(* IEC 61131-3 sources: IEC61131-3-CDSV3/Math Expressions Evaluator/src/20 Program Organization Units/Low Level, 3 files *)

(* ---- FuEvaluateExpression.pou ---- *)
(*#-#-#-#-#-#-#-#-#-#---Declaration---#-#-#-#-#-#-#-#-#-#-#-#-#*)

// Evaluates the expression.
// All expressions use LREAL as data type for operations, which is also the result output.
//
// The following math operation behaviour applies:
//  - In general: If any of the operands is a special value (+Inf, -Inf, NaN), then an error is returned
//  - For Division (/): Division by zero yields depending on ParameterList.eDivisionByZero into an error or not
//  - For Modulo (%): Both operands are converted to LINT and the result is converted back to LREAL
//
// The return value will indicate a successful evaluation.
{attribute 'qualified_only'}
FUNCTION FuEvaluateExpression : BOOL
VAR_INPUT
    typExpressionSteps: typExpressionOperationSteps;   // The expression providing steps for complex terms
    alrVariables: ARRAY [*] OF LREAL;                  // Variables to use
END_VAR
VAR_OUTPUT
    lrResult: LREAL;                                   // Result output
    sError: STRING;                                    // Error message
END_VAR
{library PRIVATE}
VAR
    i: UINT;
    tempResult: LREAL;
    tempError: STRING;

    tempInternalVariables: ARRAY [0..ParameterList.uiMaxInternalVars] OF LREAL;
END_VAR
(*#-#-#-#-#-#-#-#-#-#---Implementation---#-#-#-#-#-#-#-#-#-#-#-#-#*)

IF typExpressionSteps.uiCountSteps = 0 THEN
    FuEvaluateExpression := TRUE;
    RETURN;
END_IF

FOR i := 0 TO (typExpressionSteps.uiCountSteps - 1) BY 1 DO
    IF NOT FuEvaluateStep(typExpressionSteps.atSteps[i],  alrVariables, tempInternalVariables, lrResult => tempResult, sError => tempError) THEN
        sError := tempError;
        RETURN;
    END_IF

    // Always have the result in internal variable 0
    tempInternalVariables[0] := tempResult;

    IF
        typExpressionSteps.atSteps[i].uiInternalVariableTarget > 0 AND_THEN
        typExpressionSteps.atSteps[i].uiInternalVariableTarget >= 1 AND_THEN
        typExpressionSteps.atSteps[i].uiInternalVariableTarget <= ParameterList.uiMaxInternalVars
    THEN
        tempInternalVariables[typExpressionSteps.atSteps[i].uiInternalVariableTarget] := tempResult;
    END_IF
END_FOR

lrResult := tempResult;
FuEvaluateExpression := TRUE;

(* ---- FuStepizeExpression.pou ---- *)
(*#-#-#-#-#-#-#-#-#-#---Declaration---#-#-#-#-#-#-#-#-#-#-#-#-#*)

// Turns a tokenized expression into a stepized expression,
// providing steps for each "group" operation to be done,
// including taking care of ordering.
//
// Group operations include function calls and expressions inside ().
// Operations such as "1 + 5 - 2" are not split up and
// are evaluated left to right from the evaluator.
//
// The return value signifies whether the operation has been successfully completed.
// This function should only return false, when we run out of internal variables
// or there are no tokens.
{attribute 'qualified_only'}
FUNCTION FuStepizeExpression : BOOL
VAR_INPUT
    typTokenExpression: typTokenizedExpression;
END_VAR
VAR_OUTPUT
    typSteps: typExpressionOperationSteps;
END_VAR
{library PRIVATE}
VAR
    i: UINT;
    j: UINT;

    tempEndTokenIndex: UINT;
END_VAR
VAR // Data used throughout each loop iteration
    tempFoundGroups: ARRAY [0..ParameterList.uiMaxExpressionTokens] OF typStepizeGroupFound;
    tempCountFoundGroups: UINT;

    tempFoundGroupsTokens: ARRAY [0..ParameterList.uiMaxExpressionTokens] OF typExpressionToken;
    tempCountFoundGroupsTokens: UINT;

    tempLastStartedGroups: ARRAY [0..ParameterList.uiMaxExpressionTokens] OF UINT;
    tempCountLastStartedGroups: UINT;
END_VAR
VAR CONSTANT
    {warning disable C0228}
    INVALID_TOKEN: typExpressionToken := (eType := eTokenType.INVALID);
    EMPTY_TOKEN_ARR: ARRAY [0..ParameterList.uiMaxExpressionTokens] OF typExpressionToken;
    {warning restore C0228}
END_VAR
(*#-#-#-#-#-#-#-#-#-#---Implementation---#-#-#-#-#-#-#-#-#-#-#-#-#*)

IF typTokenExpression.uiCountTokens = 0 THEN
    RETURN;
END_IF

// Step 1: Find each group and make a list out of it
FOR i := 0 TO (typTokenExpression.uiCountTokens - 1) BY 1 DO
    IF
        typTokenExpression.atTokens[i].eType = eTokenType.GROUP_START OR_ELSE
        typTokenExpression.atTokens[i].eType = eTokenType.FUNCTION_CALL
    THEN
        tempFoundGroups[tempCountFoundGroups].uiTokenIndex := i;
        tempFoundGroups[tempCountFoundGroups].uiGroupNumber := typTokenExpression.atTokens[i].uiGroupNumber;

        tempCountFoundGroups := tempCountFoundGroups + 1;
    END_IF
END_FOR

// Skip step 2 and 3 if we found NO groups
IF tempCountFoundGroups > 0 THEN
    // Step 2: Sort the found groups array by group number and then token index
    FuInsertSortStepizeGroupFound(ADR(tempFoundGroups), tempCountFoundGroups);

    // Step 3: Consume found groups, take the tokens and insert ASSIGN_INTERNAL_VAR tokens
    //         -> Note: The found groups index + 1 corresponds to the internal variable number
    FOR i := 0 TO (tempCountFoundGroups - 1) BY 1 DO
        tempFoundGroupsTokens := EMPTY_TOKEN_ARR;
        tempCountFoundGroupsTokens := 0;

        tempCountLastStartedGroups := 0;
        tempEndTokenIndex := 0;

        FOR j := tempFoundGroups[i].uiTokenIndex TO (typTokenExpression.uiCountTokens - 1) BY 1 DO
            IF typTokenExpression.atTokens[j].eType = eTokenType.INVALID THEN
                CONTINUE;
            END_IF

            IF typTokenExpression.atTokens[j].eType = eTokenType.GROUP_START AND_THEN typTokenExpression.atTokens[j].uiGroupNumber <> tempFoundGroups[i].uiGroupNumber THEN
                // Another group started, we need to ignore those tokens now
                tempLastStartedGroups[tempCountLastStartedGroups] := typTokenExpression.atTokens[j].uiGroupNumber;
                tempCountLastStartedGroups := tempCountLastStartedGroups + 1;

                CONTINUE;
            ELSIF
                typTokenExpression.atTokens[j].eType = eTokenType.GROUP_END AND_THEN
                tempCountLastStartedGroups > 0 AND_THEN
                typTokenExpression.atTokens[j].uiGroupNumber = tempLastStartedGroups[(tempCountLastStartedGroups - 1)]
            THEN
                // Another group ended, we can now start caring again, if the count drops to 0
                tempCountLastStartedGroups := tempCountLastStartedGroups - 1;

                CONTINUE; // Taking care of using the internal variable of each group will be done later using "tempSkipTokenHints"
            ELSIF tempCountLastStartedGroups > 0 THEN
                // As long as another group are still open, prevent the other two clauses (the elsif and else) from being able to execute
                CONTINUE;
            END_IF

            IF typTokenExpression.atTokens[j].eType = eTokenType.GROUP_END AND_THEN typTokenExpression.atTokens[j].uiGroupNumber = tempFoundGroups[i].uiGroupNumber THEN
                // We've reached the end of our group, stop taking tokens away, add a hint for later about skipping tokens, and exit this loop
                tempEndTokenIndex := j;
                EXIT;
            ELSIF typTokenExpression.atTokens[j].eType = eTokenType.GROUP_START AND_THEN typTokenExpression.atTokens[j].uiGroupNumber = tempFoundGroups[i].uiGroupNumber THEN
                // Ignore group starts of ourself (we dont need those tokens)
                CONTINUE;
            END_IF

            IF typTokenExpression.atTokens[j].eType = eTokenType.FUNCTION_CALL_END AND_THEN typTokenExpression.atTokens[j].uiGroupNumber = tempFoundGroups[i].uiGroupNumber THEN
                // We've reached the end of our group, stop taking tokens away, add a hint for later about skipping tokens, and exit this loop
                tempEndTokenIndex := j;
                EXIT;
            END_IF

            tempFoundGroupsTokens[tempCountFoundGroupsTokens] := typTokenExpression.atTokens[j];
            tempCountFoundGroupsTokens := tempCountFoundGroupsTokens + 1;
        END_FOR

        typSteps.atSteps[typSteps.uiCountSteps].atTokens := tempFoundGroupsTokens;
        typSteps.atSteps[typSteps.uiCountSteps].uiCountTokens := tempCountFoundGroupsTokens;
        typSteps.atSteps[typSteps.uiCountSteps].uiInternalVariableTarget := i + 1;

        IF i >= ParameterList.uiMaxInternalVars THEN
            FuStepizeExpression := FALSE;
            RETURN;
        END_IF

        // Replace all tokens with invalid tokens, if necessary, the first token will be replaced with INTERNAL_VAR
        FOR j := tempFoundGroups[i].uiTokenIndex TO tempEndTokenIndex BY 1 DO
            typTokenExpression.atTokens[j] := INVALID_TOKEN;
        END_FOR

        IF tempFoundGroups[i].uiTokenIndex = 0 AND_THEN tempEndTokenIndex = (typTokenExpression.uiCountTokens - 1) THEN
            ;// Do not generate internal var token, because all tokens are covered
        ELSE
            // Rewrite tokens and replace them with one INTERNAL_VAR and INVALID tokens
            typTokenExpression.atTokens[tempFoundGroups[i].uiTokenIndex] := INVALID_TOKEN;
            typTokenExpression.atTokens[tempFoundGroups[i].uiTokenIndex].eType := eTokenType.INTERNAL_VAR;
            typTokenExpression.atTokens[tempFoundGroups[i].uiTokenIndex].lrValue := TO_LREAL((i + 1));
        END_IF

        typSteps.uiCountSteps := typSteps.uiCountSteps + 1;
    END_FOR
END_IF

// Step 4: Rewrite the tokens, skip INVALID tokens
FOR i := 0 TO (typTokenExpression.uiCountTokens - 1) BY 1 DO
    IF typTokenExpression.atTokens[i].eType = eTokenType.INVALID THEN
        CONTINUE;
    END_IF

    j := typSteps.atSteps[typSteps.uiCountSteps].uiCountTokens;

    typSteps.atSteps[typSteps.uiCountSteps].atTokens[j] := typTokenExpression.atTokens[i];
    typSteps.atSteps[typSteps.uiCountSteps].uiCountTokens := j + 1;
END_FOR

IF typSteps.atSteps[typSteps.uiCountSteps].uiCountTokens > 0 THEN
    typSteps.uiCountSteps := typSteps.uiCountSteps + 1;
END_IF

// Step 5: Profit, each step should now contain a particular operation set
// Note: Operations as "1 + 5 + 6" are handled inline in the evaluator, since the result of the previous op "1 + 5" can be used as "$result + 5"
FuStepizeExpression := TRUE;

(* ---- FuTokenizeExpression.pou ---- *)
(*#-#-#-#-#-#-#-#-#-#---Declaration---#-#-#-#-#-#-#-#-#-#-#-#-#*)

// Tokenizes a given math expression into a stream of tokens.
// The return value signifies whether tokenization was successful,
// or during tokenization an invalid expression was encountered.
// Please note, during tokenization not all error cases are checked.
{attribute 'qualified_only'}
FUNCTION FuTokenizeExpression : BOOL
VAR_INPUT
    sExpression: STRING(255);                 // The expression string to tokenize
END_VAR
VAR_OUTPUT
    typExpression: typTokenizedExpression;    // The tokenized expression
    sError: STRING;                           // Error message
END_VAR
{library PRIVATE}
VAR
    i: UINT;
    j: UINT;

    tempChar: BYTE;
    tempNextChar: BYTE;

    tempFunEndDetected: BOOL;
END_VAR
VAR // Data used throughout each loop iteration
    tempIndex: UINT;

    tempIdentifierStr: STRING(5);
    tempPtrByte: POINTER TO BYTE;

    tempVarOpen: BOOL;

    tempGroupOpen: INT := 0;
    tempGroupNum: UINT := 50;

    tempFunOpen: BOOL;
    tempFunIndex: UINT;
    tempFunArgsCount: UINT;

    tempNumOpen: BOOL;
    tempNumSign: BOOL; // TRUE = negative

    tempValueStr: STRING(80);
END_VAR
(*#-#-#-#-#-#-#-#-#-#---Implementation---#-#-#-#-#-#-#-#-#-#-#-#-#*)

IF sExpression = '' THEN
    sError := 'Empty expression';
    RETURN;
END_IF

sError := '';

// Assert a clean string (CODESYS does not assert that the whole string contains NUL bytes, only sets the first byte as NUL byte!)
// tempValueStr is VAR_TEMP and should get completely initialized as an empty string (all bytes = NUL), but the truth is the memory space
// gets reused and thus leftovers from the previous execution can be left there, since only the first byte is set to NUL
// (which is described by CODESYS as "new initialization", which is technically wrong!)
FOR i := 0 TO SIZEOF(tempValueStr) BY 1 DO
    tempValueStr[i] := 0;
END_FOR

FOR i := 0 TO 255 BY 1 DO
    IF sExpression[i] = 0 THEN
        EXIT;
    ELSIF tempIndex > ParameterList.uiMaxExpressionTokens THEN
        sError := 'Too many expressions';
        EXIT;
    END_IF

    tempIdentifierStr := '';
    tempPtrByte := 0;

    tempChar := sExpression[i];

    CASE tempChar OF
        Constants.CHAR_WHITESPACE, Constants.CHAR_NEWLINE, Constants.CHAR_CAR_RETURN:
            IF tempNumOpen THEN
                typExpression.atTokens[tempIndex].eType := eTokenType.NUMBER;
                typExpression.atTokens[tempIndex].lrValue := STRING_TO_LREAL(tempValueStr);

                tempValueStr := '';
                tempNumOpen := FALSE;
            ELSIF tempVarOpen THEN
                typExpression.atTokens[tempIndex].eType := eTokenType.VARIABLE;
                typExpression.atTokens[tempIndex].lrValue := STRING_TO_LREAL(tempValueStr);

                tempValueStr := '';
                tempVarOpen := FALSE;
            ELSE
                CONTINUE; // Ignore whitespace, newline (\n) and carriage return (\r)
            END_IF

        Constants.CHAR_VARIABLE:
            IF tempVarOpen OR_ELSE tempNumOpen THEN
                sError := Standard.CONCAT('Unexpected VARIABLE "\" start at token ', TO_STRING(i));
                RETURN;
            END_IF

            tempVarOpen := TRUE;
            tempValueStr := '';

            CONTINUE;

        Constants.CHAR_GROUP_START:
            tempGroupOpen := tempGroupOpen + 1;
            tempGroupNum := tempGroupNum - 1;

            typExpression.atTokens[tempIndex].eType := eTokenType.GROUP_START;
            typExpression.atTokens[tempIndex].uiGroupNumber := tempGroupNum;

        Constants.CHAR_GROUP_END:
            tempFunEndDetected := (tempFunOpen AND_THEN tempGroupNum = typExpression.atTokens[tempFunIndex].uiGroupNumber);

            IF tempNumOpen OR_ELSE tempVarOpen THEN
                typExpression.atTokens[tempIndex].eType := SEL(tempVarOpen, eTokenType.NUMBER, eTokenType.VARIABLE);
                typExpression.atTokens[tempIndex].lrValue := STRING_TO_LREAL(tempValueStr);

                tempValueStr := '';
                tempNumOpen := FALSE;
                tempVarOpen := FALSE;

                tempIndex := tempIndex + 1;
                typExpression.uiCountTokens := tempIndex;

                IF tempFunEndDetected THEN
                    tempFunArgsCount := tempFunArgsCount + 1;
                END_IF
            END_IF

            typExpression.atTokens[tempIndex].eType := SEL(tempFunEndDetected, eTokenType.GROUP_END, eTokenType.FUNCTION_CALL_END);
            typExpression.atTokens[tempIndex].uiGroupNumber := tempGroupNum;
            tempGroupNum := tempGroupNum + 1;

            IF tempFunEndDetected THEN
                // Assert for variable args functions, we have at least that many arguments,
                // or for fixed args functions, we have that many arguments as currently stored
                IF typExpression.atTokens[tempFunIndex].xArgsVariable THEN
                    IF typExpression.atTokens[tempFunIndex].uiArgsCount > tempFunArgsCount THEN
                        sError := Standard.CONCAT('Not enough arguments for variable function ', typExpression.atTokens[tempFunIndex].sIdentifier);
                        sError := Standard.CONCAT(sError, ', expected: ');
                        sError := Standard.CONCAT(sError, TO_STRING(typExpression.atTokens[tempFunIndex].uiArgsCount));
                        sError := Standard.CONCAT(sError, ', got: ');
                        sError := Standard.CONCAT(sError, TO_STRING(tempFunArgsCount));
                        RETURN;
                    END_IF
                ELSIF typExpression.atTokens[tempFunIndex].uiArgsCount <> tempFunArgsCount THEN
                    sError := Standard.CONCAT('Mismatch arguments count for function ', typExpression.atTokens[tempFunIndex].sIdentifier);
                    sError := Standard.CONCAT(sError, ', expected: ');
                    sError := Standard.CONCAT(sError, TO_STRING(typExpression.atTokens[tempFunIndex].uiArgsCount));
                    sError := Standard.CONCAT(sError, ', got: ');
                    sError := Standard.CONCAT(sError, TO_STRING(tempFunArgsCount));
                    RETURN;
                END_IF

                IF tempFunArgsCount > Constants.MAX_FUN_ARGS THEN
                    sError := Standard.CONCAT('Too many function arguments (more than ', TO_STRING(Constants.MAX_FUN_ARGS));
                    sError := Standard.CONCAT(sError, ')');
                    RETURN;
                END_IF

                typExpression.atTokens[tempFunIndex].uiArgsCount := tempFunArgsCount;

                tempFunOpen := FALSE;
                tempFunArgsCount := 0;
            ELSE
                tempGroupOpen := tempGroupOpen - 1;
            END_IF

        Constants.CHAR_COMMA:
            IF NOT tempFunOpen THEN
                sError := Standard.CONCAT('Unexpected COMMA "," outside of function at token ', TO_STRING(i));
                RETURN;
            ELSIF tempNumOpen OR_ELSE tempVarOpen THEN
                typExpression.atTokens[tempIndex].eType := SEL(tempVarOpen, eTokenType.NUMBER, eTokenType.VARIABLE);
                typExpression.atTokens[tempIndex].lrValue := STRING_TO_LREAL(tempValueStr);

                tempValueStr := '';
                tempNumOpen := FALSE;
                tempVarOpen := FALSE;

                tempIndex := tempIndex + 1;
                typExpression.uiCountTokens := tempIndex;
            END_IF

            tempFunArgsCount := tempFunArgsCount + 1;
            CONTINUE;

        Constants.CHAR_DOT:
            IF NOT tempNumOpen THEN
                sError := Standard.CONCAT('Unexpected DOT "." outside of number at token ', TO_STRING(i));
                RETURN;
            END_IF

            tempValueStr := Standard.CONCAT(tempValueStr, '.');
            CONTINUE;

        // "-" must be handled differently, as we may need to handle it as a sign
       Constants. CHAR_ADD, Constants.CHAR_SUB, Constants.CHAR_MUL,
        Constants.CHAR_DIV, Constants.CHAR_EXP, Constants.CHAR_MOD:
            IF tempNumOpen OR_ELSE tempVarOpen THEN
                typExpression.atTokens[tempIndex].eType := SEL(tempVarOpen, eTokenType.NUMBER, eTokenType.VARIABLE);
                typExpression.atTokens[tempIndex].lrValue := STRING_TO_LREAL(tempValueStr);

                tempValueStr := '';
                tempNumOpen := FALSE;
                tempVarOpen := FALSE;

                tempIndex := tempIndex + 1;
                typExpression.uiCountTokens := tempIndex;

                IF tempFunEndDetected THEN
                    tempFunArgsCount := tempFunArgsCount + 1;
                END_IF
            END_IF

            // If operator is ADD/SUB, then peek ahead to see if a number follows immediately (it's a negative number and not an operation)
            tempNextChar := sExpression[(i + 1)];
            IF
                (tempChar = Constants.CHAR_ADD OR_ELSE tempChar = Constants.CHAR_SUB) AND_THEN
                tempNextChar >= Constants.ASCII_NUM_START AND_THEN
                tempNextChar <= Constants.ASCII_NUM_END
            THEN
                tempNumOpen := TRUE;
                tempValueStr := SEL(tempChar = Constants.CHAR_ADD, '-', '');

                CONTINUE;
            END_IF

            typExpression.atTokens[tempIndex].eType := eTokenType.MATH_OP;
            typExpression.atTokens[tempIndex].sIdentifier := Util.WORD_AS_STRING(tempChar, TRUE);
    ELSE
        IF tempChar >= Constants.ASCII_NUM_START AND_THEN tempChar <= Constants.ASCII_NUM_END THEN
            IF NOT tempVarOpen AND_THEN NOT tempNumOpen THEN
                tempNumOpen := TRUE;
                tempValueStr := '';
            END_IF

            tempValueStr := Standard.CONCAT(tempValueStr, TO_STRING((tempChar - Constants.ASCII_NUM_START)));
            CONTINUE;
        ELSIF tempChar >= Constants.ASCII_ALPHA_START AND_THEN tempChar <= Constants.ASCII_ALPHA_END THEN
            // We can not call a function inside a function
            IF tempFunOpen THEN
                sError := Standard.CONCAT('Nested function calls are not supported, found at token ', TO_STRING(i));
                RETURN;
            END_IF

            FOR j := i TO (i + 5) BY 1 DO
                IF sExpression[j] = Constants.CHAR_GROUP_START THEN
                    EXIT;
                END_IF

                tempIdentifierStr[(j - i)] := sExpression[j];

                // Assert string is correctly NUL terminated (prevent "MAXIN" when first "LIMIT" and then "MAX" was tokenized)
                tempIdentifierStr[(j - i + 1)] := 0;
            END_FOR

            i := j - 1;

            IF
                tempIdentifierStr = Constants.FUN_ABS OR_ELSE
                tempIdentifierStr = Constants.FUN_ACOS OR_ELSE
                tempIdentifierStr = Constants.FUN_ASIN OR_ELSE
                tempIdentifierStr = Constants.FUN_ATAN OR_ELSE
                tempIdentifierStr = Constants.FUN_CEIL OR_ELSE
                tempIdentifierStr = Constants.FUN_COS OR_ELSE
                tempIdentifierStr = Constants.FUN_DEG OR_ELSE
                tempIdentifierStr = Constants.FUN_FLOOR OR_ELSE
                tempIdentifierStr = Constants.FUN_LOG OR_ELSE
                tempIdentifierStr = Constants.FUN_LN OR_ELSE
                tempIdentifierStr = Constants.FUN_RAD OR_ELSE
                tempIdentifierStr = Constants.FUN_ROUND OR_ELSE
                tempIdentifierStr = Constants.FUN_SIN OR_ELSE
                tempIdentifierStr = Constants.FUN_SQRT OR_ELSE
                tempIdentifierStr = Constants.FUN_TAN
            THEN
                // Single arg functions
                typExpression.atTokens[tempIndex].uiArgsCount := 1;
            ELSIF
                tempIdentifierStr = Constants.FUN_TRUNC
            THEN
                // Dual arg functions
                typExpression.atTokens[tempIndex].uiArgsCount := 2;
            ELSIF
                tempIdentifierStr = Constants.FUN_LIMIT
            THEN
                // Triple arg functions
                typExpression.atTokens[tempIndex].uiArgsCount := 3;
            ELSIF
                tempIdentifierStr = Constants.FUN_AVGA OR_ELSE
                tempIdentifierStr = Constants.FUN_MAX OR_ELSE
                tempIdentifierStr = Constants.FUN_MIN
            THEN
                // Variable arg functions (at least 2)
                typExpression.atTokens[tempIndex].uiArgsCount := 2;
                typExpression.atTokens[tempIndex].xArgsVariable := TRUE;
            ELSE
                // Invalid function name
                sError := Standard.CONCAT('Unknown function ', tempIdentifierStr);
                RETURN;
            END_IF

            // Peek at the next expression token and check if it's a GROUP_START token
            IF sExpression[(i + 1)] <> Constants.CHAR_GROUP_START THEN
                // If not, invalid expression
                sError := Standard.CONCAT('Expected GROUP_START "(" for function call at token ', TO_STRING((i + 1)));
                RETURN;
            END_IF

            // Skip next token, as we've already consumed it
            i := i + 1;

            tempFunIndex := tempIndex;
            tempGroupNum := tempGroupNum - 1;

            typExpression.atTokens[tempIndex].eType := eTokenType.FUNCTION_CALL;
            typExpression.atTokens[tempIndex].sIdentifier := tempIdentifierStr;
            typExpression.atTokens[tempIndex].uiGroupNumber := tempGroupNum;

            tempFunOpen := TRUE;
            tempFunArgsCount := 0;
        ELSE
            // Invalid expression
            sError := Standard.CONCAT('Invalid character at token ', TO_STRING(i));
            RETURN;
        END_IF
    END_CASE

    tempIndex := tempIndex + 1;
    typExpression.uiCountTokens := tempIndex;
END_FOR

// If var or num open, close it and append as token
IF tempVarOpen THEN
    typExpression.atTokens[tempIndex].eType := eTokenType.VARIABLE;
    typExpression.atTokens[tempIndex].lrValue := STRING_TO_LREAL(tempValueStr);

    tempIndex := tempIndex + 1;
ELSIF tempNumOpen THEN
    typExpression.atTokens[tempIndex].eType := eTokenType.NUMBER;
    typExpression.atTokens[tempIndex].lrValue := STRING_TO_LREAL(tempValueStr);

    tempIndex := tempIndex + 1;
END_IF

typExpression.uiCountTokens := tempIndex;
FuTokenizeExpression := (tempIndex > 0 AND_THEN NOT tempVarOpen AND_THEN tempGroupOpen = 0 AND_THEN NOT tempFunOpen);
